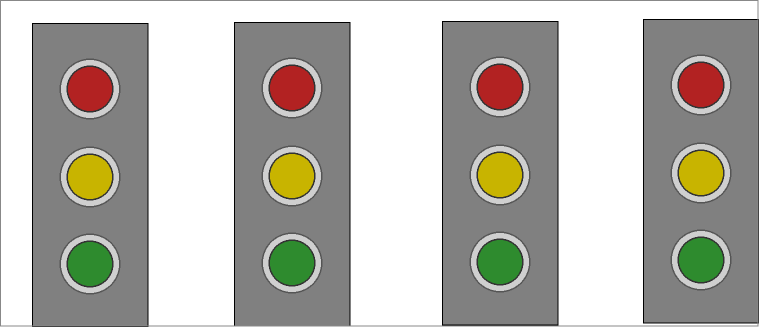
VISUALIZATION visuTrafficLights  // 759x327
    RoundedRectangle (32,23 116x304), invisible if: MAIN.fbTrafficLightController.arTrafficLightsInvisible[1]
    Lamp1 (55,54 70x70), variable: MAIN.fbTrafficLightController.arTrafficLights[1].RedLight, invisible if: MAIN.fbTrafficLightController.arTrafficLightsInvisible[1], style: Lamp-Lamp1-Red
    Lamp1 (55,142 70x70), variable: MAIN.fbTrafficLightController.arTrafficLights[1].YellowLight, invisible if: MAIN.fbTrafficLightController.arTrafficLightsInvisible[1], style: Lamp-Lamp1-Yellow
    Lamp1 (55,229 70x70), variable: MAIN.fbTrafficLightController.arTrafficLights[1].GreenLight, invisible if: MAIN.fbTrafficLightController.arTrafficLightsInvisible[1], style: Lamp-Lamp1-Green
    RoundedRectangle (234,22 116x304), invisible if: MAIN.fbTrafficLightController.arTrafficLightsInvisible[2]
    Lamp1 (257,53 70x70), variable: MAIN.fbTrafficLightController.arTrafficLights[2].RedLight, invisible if: MAIN.fbTrafficLightController.arTrafficLightsInvisible[2], style: Lamp-Lamp1-Red
    Lamp1 (257,141 70x70), variable: MAIN.fbTrafficLightController.arTrafficLights[2].YellowLight, invisible if: MAIN.fbTrafficLightController.arTrafficLightsInvisible[2], style: Lamp-Lamp1-Yellow
    Lamp1 (257,228 70x70), variable: MAIN.fbTrafficLightController.arTrafficLights[2].GreenLight, invisible if: MAIN.fbTrafficLightController.arTrafficLightsInvisible[2], style: Lamp-Lamp1-Green
    RoundedRectangle (442,21 116x304), invisible if: MAIN.fbTrafficLightController.arTrafficLightsInvisible[3]
    Lamp1 (465,52 70x70), variable: MAIN.fbTrafficLightController.arTrafficLights[3].RedLight, invisible if: MAIN.fbTrafficLightController.arTrafficLightsInvisible[3], style: Lamp-Lamp1-Red
    Lamp1 (465,140 70x70), variable: MAIN.fbTrafficLightController.arTrafficLights[3].YellowLight, invisible if: MAIN.fbTrafficLightController.arTrafficLightsInvisible[3], style: Lamp-Lamp1-Yellow
    Lamp1 (465,227 70x70), variable: MAIN.fbTrafficLightController.arTrafficLights[3].GreenLight, invisible if: MAIN.fbTrafficLightController.arTrafficLightsInvisible[3], style: Lamp-Lamp1-Green
    RoundedRectangle (643,19 116x304), invisible if: MAIN.fbTrafficLightController.arTrafficLightsInvisible[4]
    Lamp1 (666,50 70x70), variable: MAIN.fbTrafficLightController.arTrafficLights[4].RedLight, invisible if: MAIN.fbTrafficLightController.arTrafficLightsInvisible[4], style: Lamp-Lamp1-Red
    Lamp1 (666,138 70x70), variable: MAIN.fbTrafficLightController.arTrafficLights[4].YellowLight, invisible if: MAIN.fbTrafficLightController.arTrafficLightsInvisible[4], style: Lamp-Lamp1-Yellow
    Lamp1 (666,225 70x70), variable: MAIN.fbTrafficLightController.arTrafficLights[4].GreenLight, invisible if: MAIN.fbTrafficLightController.arTrafficLightsInvisible[4], style: Lamp-Lamp1-Green
END_VISUALIZATION

(* stored: Version 1.1.0.1, ProductVersion 3.1.4024.12
   Visu visuTrafficLights: Id {8d66701b-744a-426f-a33f-cb044005c6fe} *)
